// Mitsubishi GX Works2 project: 타이머   PLC: Q02/Q02H

PROGRAM MAIN
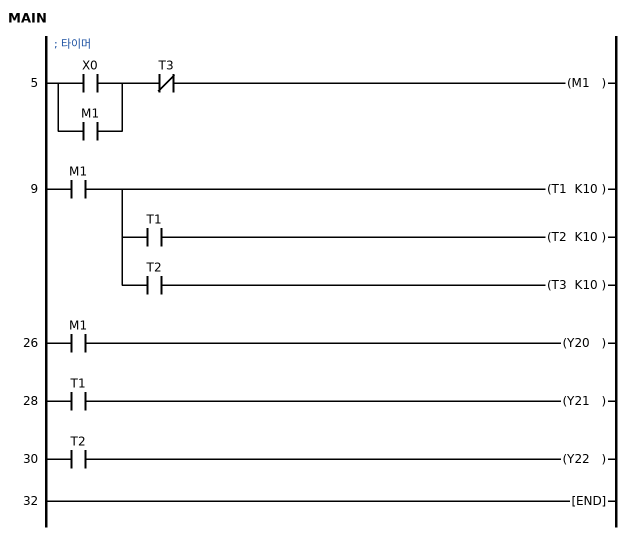
; 타이머
5     LD      X0
      OR      M1
      ANI     T3
      OUT     M1
9     LD      M1
      OUT     T1 K10
      MPS
      AND     T1
      OUT     T2 K10
      MPP
      AND     T2
      OUT     T3 K10
26    LD      M1
      OUT     Y20
28    LD      T1
      OUT     Y21
30    LD      T2
      OUT     Y22
32    END
END_PROGRAM
